Fanuc KAREL source: wtimeshift.kl

PROGRAM wtimeshift
%NOLOCKGROUP
VAR
  p : POSITION
  q : POSITION
  i : INTEGER
  r : REAL
BEGIN
  WITH $TIME_SHIFT = 10 MOVE TO p
END wtimeshift
